PROGRAM RFID_FB
VAR
	RFID_FB:							FB_BIS00LH;
	RFID_IO:							ST_BIS00LH_IO;	

END_VAR

RFID_FB(IO := RFID_IO);

END_PROGRAM

(* stored: Version 1.1.0.1, ProductVersion 3.1.4022.12
   POU RFID_FB: Id {650786ac-352d-4cae-a096-3d6b11d9e03e}, SpecialFunc None *)
